PROGRAM P_Demo_FB_HVACMotor3Speed
VAR
    fb : FB_HVACMotor3Speed;                            // 被演示 FB 实例
    eDataSecurityType_in : E_HVACDataSecurityType ;
    bSetDefault_in : BOOL := FALSE;
    bEnable_in : BOOL := FALSE;
    bAutoSpeed1_in : BOOL := FALSE;
    bAutoSpeed2_in : BOOL := FALSE;
    bAutoSpeed3_in : BOOL := FALSE;
    eCtrlModeActuator_in : E_HVACActuatorMode ;
    bMotorProtecSpeed1_in : BOOL := FALSE;
    bMotorProtecSpeed2_in : BOOL := FALSE;
    bMotorProtecSpeed3_in : BOOL := FALSE;
    bFeedbContactorSpeed1_in : BOOL := FALSE;
    bFeedbContactorSpeed2_in : BOOL := FALSE;
    bFeedbContactorSpeed3_in : BOOL := FALSE;
    bFeedbProcess_in : BOOL := FALSE;
    bRepairSwitch_in : BOOL := FALSE;
    bManSwitch_in : BOOL := FALSE;
    bCtrlVoltage_in : BOOL := FALSE;
    bReset_in : BOOL := FALSE;
    tStartDelay_io : TIME := T#0S;
    tStopDelay_io : TIME := T#0S;
    tDelayFeedbContactorSpeed1_io : TIME := T#0S;
    tDelayFeedbContactorSpeed2_io : TIME := T#0S;
    tDelayFeedbContactorSpeed3_io : TIME := T#0S;
    tFeedbProcessTimer_io : TIME := T#0S;
    tDelayFeedbProcess_io : TIME := T#0S;
    tDelaySpeed1_io : TIME := T#0S;
    tDelaySpeed2_io : TIME := T#0S;
    tDelaySpeed1ToSpeed2ToSpeed3_io : TIME := T#0S;
    tDelaySpeed2ToSpeed1_io : TIME := T#0S;
    tDelaySpeed3ToSpeed2_io : TIME := T#0S;
    bMotorSpeed1_out : BOOL;
    bMotorSpeed2_out : BOOL;
    bMotorSpeed3_out : BOOL;
    wState_out : WORD;
    bStateAutoSpeed1_out : BOOL;
    bStateAutoSpeed2_out : BOOL;
    bStateAutoSpeed3_out : BOOL;
    bStateRepairSwitch_out : BOOL;
    bStateManSwitch_out : BOOL;
    eStateModeActuator_out : E_HVACActuatorMode;
    bErrorGeneral_out : BOOL;
    wError_out : WORD;
    bErrorMotorprotecSpeed1_out : BOOL;
    bErrorMotorprotecSpeed2_out : BOOL;
    bErrorMotorprotecSpeed3_out : BOOL;
    bErrorFeedbContactorSpeed1_out : BOOL;
    bErrorFeedbContactorSpeed2_out : BOOL;
    bErrorFeedbContactorSpeed3_out : BOOL;
    bErrorFeedbProcess_out : BOOL;
    bInvalidParameter_out : BOOL;
END_VAR

// ============================================================================
// Tc2_HVAC.FB_HVACMotor3Speed 演示程序
// ============================================================================
// 场景：把本 FB 实例化到一个 PLC 程序里，每周期单次调用；按需要把 VAR_INPUT 与
//       VAR_IN_OUT 接到工程信号；VAR_OUTPUT 写入对应监视变量。
// 价值：使用本 FB 比手写状态机 / 控制算法节省大量代码；与 Tc2_HVAC 体系内其它 FB
//       直接对接，命名 / 持久化 / 模式仲裁等约定一致。具体语义见 FB_HVACMotor3Speed.md 主文档。
// 验证步骤：
//   1. 右键 PLC 项目下 POUs 文件夹 → Add → Existing Item → 选本 .TcPOU 文件
//   2. 引用 Tc2_HVAC（References → Add library）
//   3. 编译 → 登录 → 运行
//   4. 在线写各 *_in 输入信号触发 FB；在线 monitor *_out 引脚观察状态
// ============================================================================

fb(
    eDataSecurityType := eDataSecurityType_in,
    bSetDefault := bSetDefault_in,
    bEnable := bEnable_in,
    bAutoSpeed1 := bAutoSpeed1_in,
    bAutoSpeed2 := bAutoSpeed2_in,
    bAutoSpeed3 := bAutoSpeed3_in,
    eCtrlModeActuator := eCtrlModeActuator_in,
    bMotorProtecSpeed1 := bMotorProtecSpeed1_in,
    bMotorProtecSpeed2 := bMotorProtecSpeed2_in,
    bMotorProtecSpeed3 := bMotorProtecSpeed3_in,
    bFeedbContactorSpeed1 := bFeedbContactorSpeed1_in,
    bFeedbContactorSpeed2 := bFeedbContactorSpeed2_in,
    bFeedbContactorSpeed3 := bFeedbContactorSpeed3_in,
    bFeedbProcess := bFeedbProcess_in,
    bRepairSwitch := bRepairSwitch_in,
    bManSwitch := bManSwitch_in,
    bCtrlVoltage := bCtrlVoltage_in,
    bReset := bReset_in,
    tStartDelay := tStartDelay_io,
    tStopDelay := tStopDelay_io,
    tDelayFeedbContactorSpeed1 := tDelayFeedbContactorSpeed1_io,
    tDelayFeedbContactorSpeed2 := tDelayFeedbContactorSpeed2_io,
    tDelayFeedbContactorSpeed3 := tDelayFeedbContactorSpeed3_io,
    tFeedbProcessTimer := tFeedbProcessTimer_io,
    tDelayFeedbProcess := tDelayFeedbProcess_io,
    tDelaySpeed1 := tDelaySpeed1_io,
    tDelaySpeed2 := tDelaySpeed2_io,
    tDelaySpeed1ToSpeed2ToSpeed3 := tDelaySpeed1ToSpeed2ToSpeed3_io,
    tDelaySpeed2ToSpeed1 := tDelaySpeed2ToSpeed1_io,
    tDelaySpeed3ToSpeed2 := tDelaySpeed3ToSpeed2_io,
    bMotorSpeed1 => bMotorSpeed1_out,
    bMotorSpeed2 => bMotorSpeed2_out,
    bMotorSpeed3 => bMotorSpeed3_out,
    wState => wState_out,
    bStateAutoSpeed1 => bStateAutoSpeed1_out,
    bStateAutoSpeed2 => bStateAutoSpeed2_out,
    bStateAutoSpeed3 => bStateAutoSpeed3_out,
    bStateRepairSwitch => bStateRepairSwitch_out,
    bStateManSwitch => bStateManSwitch_out,
    eStateModeActuator => eStateModeActuator_out,
    bErrorGeneral => bErrorGeneral_out,
    wError => wError_out,
    bErrorMotorprotecSpeed1 => bErrorMotorprotecSpeed1_out,
    bErrorMotorprotecSpeed2 => bErrorMotorprotecSpeed2_out,
    bErrorMotorprotecSpeed3 => bErrorMotorprotecSpeed3_out,
    bErrorFeedbContactorSpeed1 => bErrorFeedbContactorSpeed1_out,
    bErrorFeedbContactorSpeed2 => bErrorFeedbContactorSpeed2_out,
    bErrorFeedbContactorSpeed3 => bErrorFeedbContactorSpeed3_out,
    bErrorFeedbProcess => bErrorFeedbProcess_out,
    bInvalidParameter => bInvalidParameter_out
);

END_PROGRAM

(* stored: Version 1.1.0.1, ProductVersion 3.1.4024.5
   POU P_Demo_FB_HVACMotor3Speed: Id {721fcc4d-0c67-5484-a948-86275a5369d8}, SpecialFunc None *)
